FUNCTION_BLOCK ResolveTestBasicFbt
END_FUNCTION_BLOCK
